# EPICS autosave request: iocs/softDetectorIOC/iocBoot/iocSoftDetector/auto_settings.req
file "softDetector_settings.req",    P=$(P),  R=cam1:
file "softDetector_settings.req",    P=$(P),  R=cam2:
file "NDStdArrays_settings.req",    P=$(P),  R=image1:
file "commonPlugin_settings.req",   P=$(P)
